FUNCTION_BLOCK FB_PFCA7 EXTENDS ZigaLibs_IoLink.FB_IoLinkState IMPLEMENTS I_PFCA7
VAR
	InputProcessData	AT %I* : ST_PFCA7_InputProcessData;
	OutputProcessData	AT %Q* : ST_PFCA7_OutputProcessData;
	_inputProcessData	: ST_PFCA7_InputProcessData;
	_maxFlow			: REAL;
	_measuredFlow		: REAL;
	_IoLinkMaxFlowValue	: INT := 4_000;
END_VAR

(* Should be called cyclically to execute necesary calls
 This is used instead of FBXXX() -> FBXXX.Execute() and makes the programming more consistent.*)
METHOD Execute
VAR_INPUT
	bEnable			: BOOL;	// Enable flow setting
	fFlowSetpoint	: REAL;	// Flow setpoint
END_VAR
_inputProcessData := InputProcessData;

// Flow measurement
_measuredFlow := _maxFlow * (1.0 * InputProcessData.MeasuredFlow)/INT_TO_REAL(_IoLinkMaxFlowValue);

// Output section
IF bEnable = FALSE OR _maxFlow = 0 THEN
	OutputProcessData.CommandedFlowRate := 0;
ELSE
	OutputProcessData.CommandedFlowRate := REAL_TO_UINT((INT_TO_REAL(_IoLinkMaxFlowValue) * MIN(fFlowSetpoint, _maxFlow)/_maxFlow));
END_IF
END_METHOD

METHOD FB_init : BOOL
VAR_INPUT
	bInitRetains : BOOL; // if TRUE, the retain variables are initialized (warm start / cold start)
	bInCopyCode : BOOL;  // if TRUE, the instance afterwards gets moved into the copy code (online change)
	logger		: REFERENCE TO ZigaLibs_Logging.I_Logger;
	fMaxFlow	: REAL;
END_VAR
_maxFlow := fMaxFlow;
END_METHOD

 {attribute 'monitoring' := 'variable'}
// Gets device feedback structure
PROPERTY PUBLIC Feedback : REFERENCE TO ST_PFCA7_InputProcessData
GET
Feedback REF= _inputProcessData;
END_GET
END_PROPERTY

(* Gets or sets the IO link max flow value, this is used for value scaling and should be read from the datasheet.*)
PROPERTY IoLinkMaxFlowValue : INT
GET
IoLinkMaxFlowValue := _IoLinkMaxFlowValue;
END_GET
SET
_IoLinkMaxFlowValue := IoLinkMaxFlowValue;
END_SET
END_PROPERTY

(* Gets or sets the max flow*)
PROPERTY MaxFlow : REAL
GET
MaxFlow := _maxFlow;
END_GET
SET
_maxFlow := MaxFlow;
END_SET
END_PROPERTY

(* Gets the measured flow*)
PROPERTY MeasuredFlow : REAL
GET
MeasuredFlow := _measuredFlow;
END_GET
END_PROPERTY

END_FUNCTION_BLOCK

(* stored: Version 1.1.0.1, ProductVersion 3.1.4024.16
   POU FB_PFCA7: Id {8dc9b630-9794-007d-3de2-519416ea1546}, SpecialFunc None
   Folder Constructor: Id {64f0e145-4ac8-0d45-1410-db2549bf3417}
   Folder Methods - public: Id {cfb36886-264c-0650-3711-598c6c8980c1}
   Folder Properties - public: Id {bb41fb88-9325-041c-310e-5aeac7d846df}
   Method Execute: Id {98911978-17e7-0fac-36eb-c126d3cbf294}
   Method FB_init: Id {8e7bf8cf-dc2c-0203-2302-a00d8b13199a}
   Property Feedback: Id {44cd6220-fbd9-01a3-185d-6873e34156c6}
   Get Get: Id {41876fe9-303e-0fe5-1172-a8667fd47740}
   Property IoLinkMaxFlowValue: Id {e06e514d-6363-0830-0dbd-7ce5f9e8db10}
   Get Get: Id {86aeeebb-97e6-0af8-2f0d-de85513df84e}
   Set Set: Id {34a96f17-1f32-03d5-3f85-0a65efdde3d9}
   Property MaxFlow: Id {4cbd69d9-19ff-052a-3942-88e3c71e2a38}
   Get Get: Id {99a67f22-17bd-0d21-35dd-68d22110ac80}
   Set Set: Id {c134333e-b11f-009d-164c-6bdbdd6230af}
   Property MeasuredFlow: Id {acee1752-1f59-0501-089a-494f62884bde}
   Get Get: Id {a2ff2a66-19f9-0f3a-3610-05afb6f4bf41} *)
